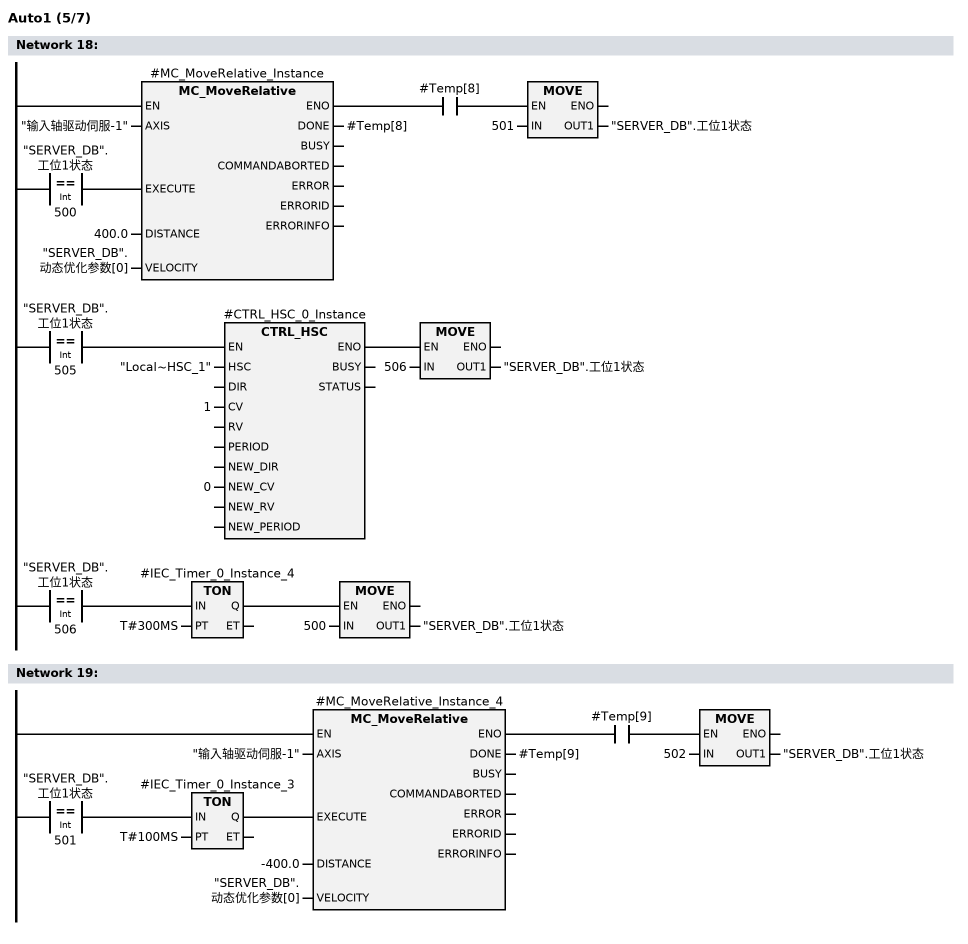
   // ENO of a box is taken as its EN; it also drops when the box reports an error
   #MC_MoveRelative_Instance(Axis := "输入轴驱动伺服-1",   // MC_MoveRelative
                           Execute := "SERVER_DB".工位1状态 = 500,
                           Distance := 400.0,
                           Velocity := "SERVER_DB".动态优化参数[0],
                           Done => #Temp[8]);
   IF #Temp[8] THEN "SERVER_DB".工位1状态 := 501; END_IF;
   #_w1 := "SERVER_DB".工位1状态 = 505;
   IF #_w1 THEN
       #CTRL_HSC_0_Instance(HSC := "Local~HSC_1", CV := 1, NEW_CV := 0);   // CTRL_HSC
       "SERVER_DB".工位1状态 := 506;
   END_IF;
   #IEC_Timer_0_Instance_4(IN := "SERVER_DB".工位1状态 = 506, PT := T#300MS);   // TON
   IF #IEC_Timer_0_Instance_4.Q THEN "SERVER_DB".工位1状态 := 500; END_IF;
END_REGION

REGION Network 19
   // ENO of a box is taken as its EN; it also drops when the box reports an error
   #IEC_Timer_0_Instance_3(IN := "SERVER_DB".工位1状态 = 501, PT := T#100MS);   // TON
   #MC_MoveRelative_Instance_4(Axis := "输入轴驱动伺服-1",   // MC_MoveRelative
                           Execute := #IEC_Timer_0_Instance_3.Q,
                           Distance := -400.0,
                           Velocity := "SERVER_DB".动态优化参数[0],
                           Done => #Temp[9]);
   IF #Temp[9] THEN "SERVER_DB".工位1状态 := 502; END_IF;
END_REGION

REGION Network 20
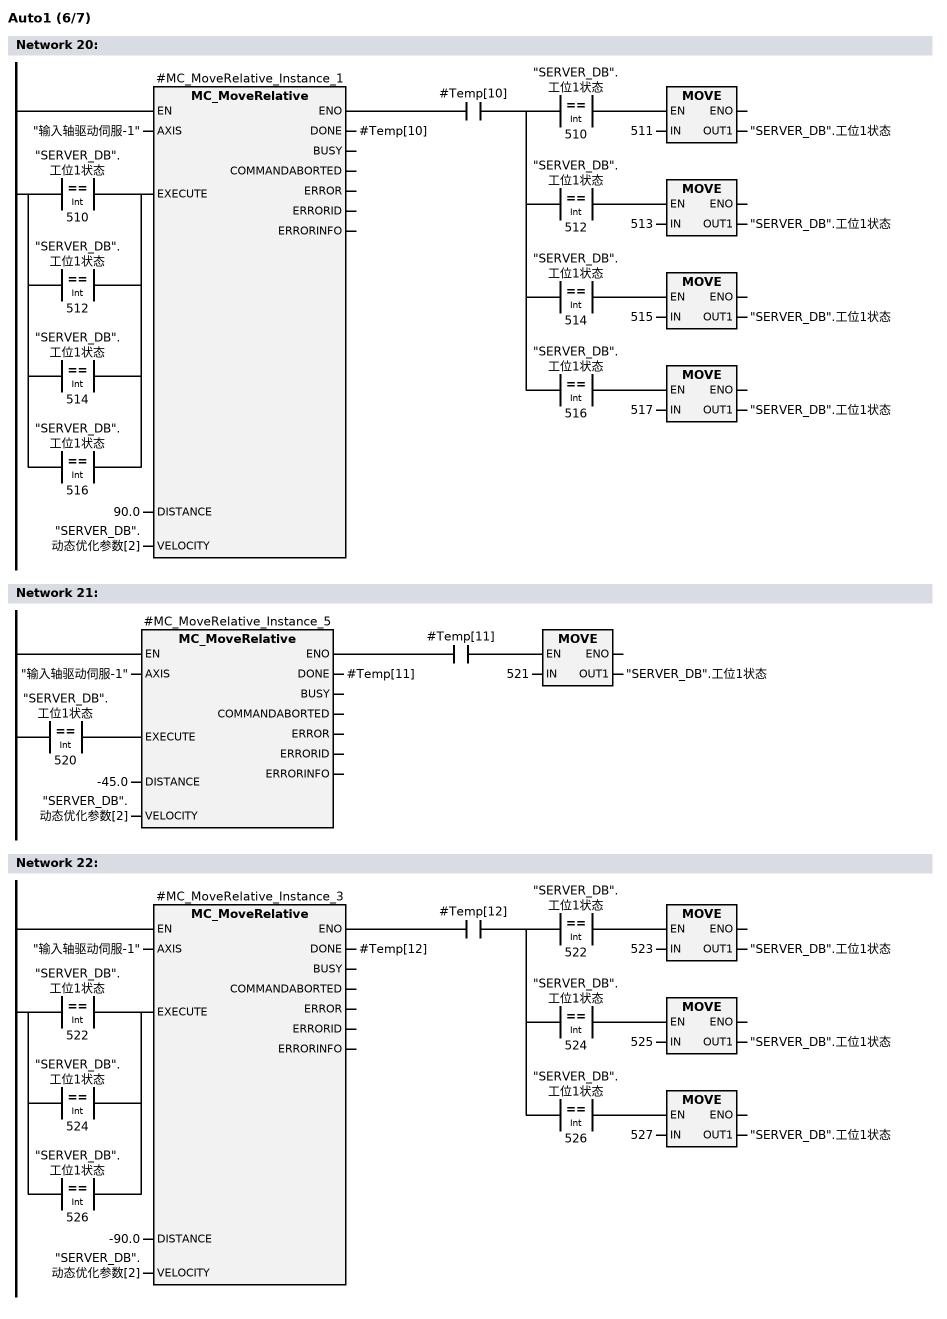
   // ENO of a box is taken as its EN; it also drops when the box reports an error
   #MC_MoveRelative_Instance_1(Axis := "输入轴驱动伺服-1",   // MC_MoveRelative
                           Execute := ("SERVER_DB".工位1状态 = 510) OR ("SERVER_DB".工位1状态 = 512) OR ("SERVER_DB".工位1状态 = 514) OR ("SERVER_DB".工位1状态 = 516),
                           Distance := 90.0,
                           Velocity := "SERVER_DB".动态优化参数[2],
                           Done => #Temp[10]);
   IF #Temp[10] AND ("SERVER_DB".工位1状态 = 510) THEN "SERVER_DB".工位1状态 := 511; END_IF;
   IF #Temp[10] AND ("SERVER_DB".工位1状态 = 512) THEN "SERVER_DB".工位1状态 := 513; END_IF;
   IF #Temp[10] AND ("SERVER_DB".工位1状态 = 514) THEN "SERVER_DB".工位1状态 := 515; END_IF;
   IF #Temp[10] AND ("SERVER_DB".工位1状态 = 516) THEN "SERVER_DB".工位1状态 := 517; END_IF;
END_REGION

REGION Network 21
   // ENO of a box is taken as its EN; it also drops when the box reports an error
   #MC_MoveRelative_Instance_5(Axis := "输入轴驱动伺服-1",   // MC_MoveRelative
                           Execute := "SERVER_DB".工位1状态 = 520,
                           Distance := -45.0,
                           Velocity := "SERVER_DB".动态优化参数[2],
                           Done => #Temp[11]);
   IF #Temp[11] THEN "SERVER_DB".工位1状态 := 521; END_IF;
END_REGION

REGION Network 22
   // ENO of a box is taken as its EN; it also drops when the box reports an error
   #MC_MoveRelative_Instance_3(Axis := "输入轴驱动伺服-1",   // MC_MoveRelative
                           Execute := ("SERVER_DB".工位1状态 = 522) OR ("SERVER_DB".工位1状态 = 524) OR ("SERVER_DB".工位1状态 = 526),
                           Distance := -90.0,
                           Velocity := "SERVER_DB".动态优化参数[2],
                           Done => #Temp[12]);
   IF #Temp[12] AND ("SERVER_DB".工位1状态 = 522) THEN "SERVER_DB".工位1状态 := 523; END_IF;
   IF #Temp[12] AND ("SERVER_DB".工位1状态 = 524) THEN "SERVER_DB".工位1状态 := 525; END_IF;
   IF #Temp[12] AND ("SERVER_DB".工位1状态 = 526) THEN "SERVER_DB".工位1状态 := 527; END_IF;
END_REGION

REGION Network 23
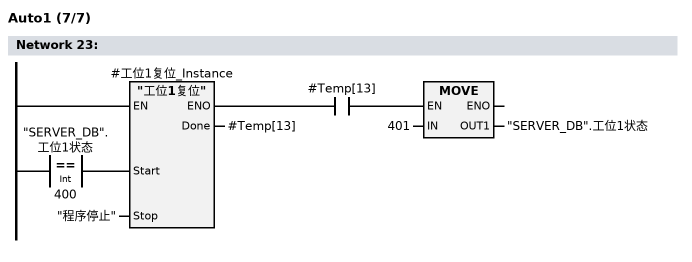
   RUNG wire#powerrail
      #工位1复位_Instance(Start := wire#w1, Stop := "程序停止", Done => #Temp[13])
      Contact( #Temp[13] )
      Move(in := 401, out1 => "SERVER_DB".工位1状态)
   END_RUNG
   RUNG wire#powerrail
      { S7_Templates := "SrcType := Int" } EQ_Contact(in1 := "SERVER_DB".工位1状态, in2 := 400)
   END_RUNG wire#w1
   // the same network as SCL:
   #工位1复位_Instance(Start := "SERVER_DB".工位1状态 = 400, Stop := "程序停止", Done => #Temp[13], ENO => #_w1);   // "工位1复位"
   IF #_w1 AND #Temp[13] THEN "SERVER_DB".工位1状态 := 401; END_IF;
END_REGION
END_FUNCTION_BLOCK

FUNCTION_BLOCK "输入轴二次夹紧"   // FB10, LAD
{ S7_Optimized_Access := 'TRUE' }
VERSION : 0.1
   VAR_INPUT
      Axis : TO_PositioningAxis;
      Start : Bool;
      夹紧位置 : Real;
   END_VAR
   VAR_OUTPUT
      Done : Bool;
   END_VAR
   VAR
      "Step" : Int;
      Temp : Array[0..3] of Bool;
      MC_MoveAbsolute_Instance : MC_MoveAbsolute;
      IEC_Timer_0_Instance : TON_TIME;
      IEC_Timer_0_Instance_1 : TON_TIME;
   END_VAR
   VAR_TEMP   // added for the SCL form of the ladder/FBD networks
      _w1 : Bool;
   END_VAR
BEGIN

REGION Network 1
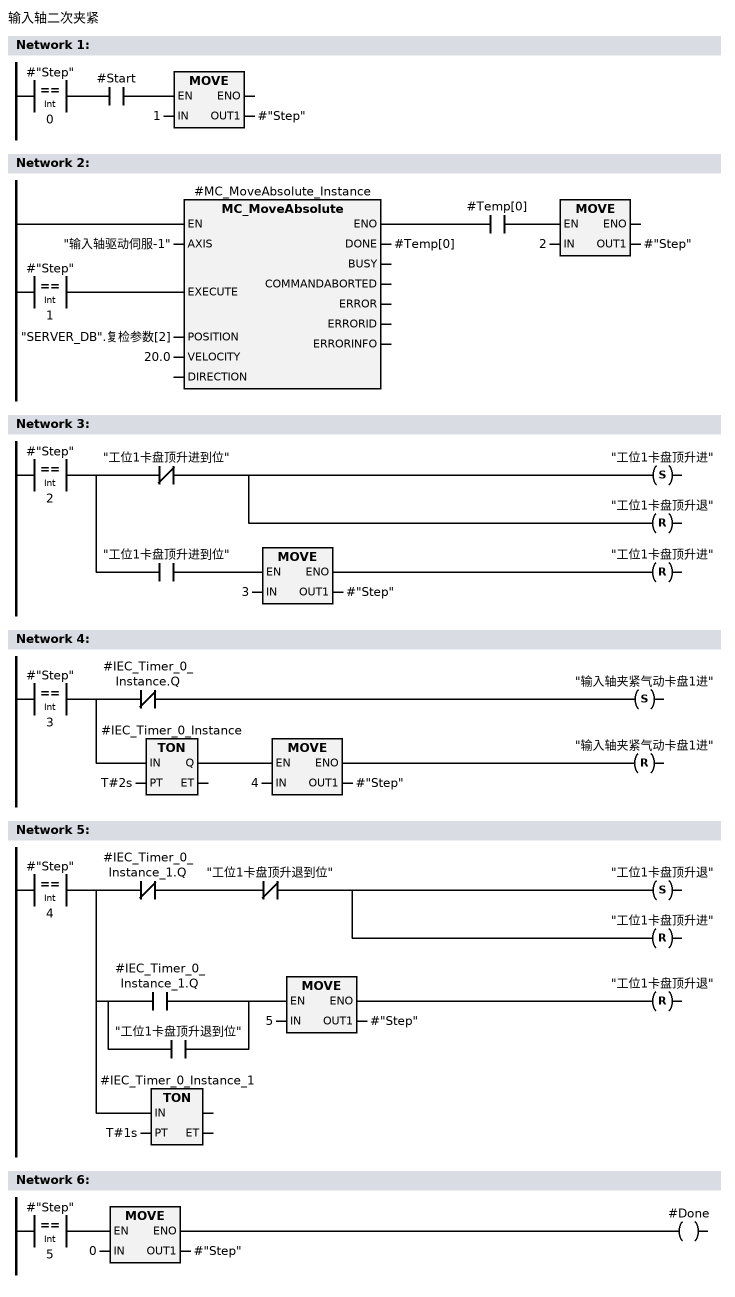
   RUNG wire#powerrail
      { S7_Templates := "SrcType := Int" } EQ_Contact(in1 := #"Step", in2 := 0)
      Contact( #Start )
      Move(in := 1, out1 => #"Step")
   END_RUNG
   // the same network as SCL:
   IF (#"Step" = 0) AND #Start THEN #"Step" := 1; END_IF;
END_REGION

REGION Network 2
   // ENO of a box is taken as its EN; it also drops when the box reports an error
   #MC_MoveAbsolute_Instance(Axis := "输入轴驱动伺服-1",   // MC_MoveAbsolute
                           Execute := #"Step" = 1,
                           Position := "SERVER_DB".复检参数[2],
                           Velocity := 20.0,
                           Done => #Temp[0]);
   IF #Temp[0] THEN #"Step" := 2; END_IF;
END_REGION

REGION Network 3
   RUNG wire#powerrail
      { S7_Templates := "SrcType := Int" } EQ_Contact(in1 := #"Step", in2 := 2)
      wire#w1
      I_Contact( "工位1卡盘顶升进到位" )
      wire#w2
      S_Coil( "工位1卡盘顶升进" )
   END_RUNG
   RUNG wire#w2
      R_Coil( "工位1卡盘顶升退" )
   END_RUNG
   RUNG wire#w1
      Contact( "工位1卡盘顶升进到位" )
      Move(in := 3, out1 => #"Step")
      R_Coil( "工位1卡盘顶升进" )
   END_RUNG
   // the same network as SCL:
   #_w1 := #"Step" = 2;
   IF #_w1 AND NOT "工位1卡盘顶升进到位" THEN
       "工位1卡盘顶升进" := TRUE;
       "工位1卡盘顶升退" := FALSE;
   END_IF;
   IF #_w1 AND "工位1卡盘顶升进到位" THEN
       #"Step" := 3;
       "工位1卡盘顶升进" := FALSE;
   END_IF;
END_REGION

REGION Network 4
   #_w1 := #"Step" = 3;
   IF #_w1 AND NOT #IEC_Timer_0_Instance.Q THEN "输入轴夹紧气动卡盘1进" := TRUE; END_IF;
   #IEC_Timer_0_Instance(IN := #_w1, PT := T#2s);   // TON
   IF #IEC_Timer_0_Instance.Q THEN
       #"Step" := 4;
       "输入轴夹紧气动卡盘1进" := FALSE;
   END_IF;
END_REGION

REGION Network 5
   #_w1 := #"Step" = 4;
   IF #_w1 AND NOT #IEC_Timer_0_Instance_1.Q AND NOT "工位1卡盘顶升退到位" THEN
       "工位1卡盘顶升退" := TRUE;
       "工位1卡盘顶升进" := FALSE;
   END_IF;
   IF #_w1 AND (#IEC_Timer_0_Instance_1.Q OR "工位1卡盘顶升退到位") THEN
       #"Step" := 5;
       "工位1卡盘顶升退" := FALSE;
   END_IF;
   #IEC_Timer_0_Instance_1(IN := #_w1, PT := T#1s);   // TON
END_REGION

REGION Network 6
   RUNG wire#powerrail
      { S7_Templates := "SrcType := Int" } EQ_Contact(in1 := #"Step", in2 := 5)
      Move(in := 0, out1 => #"Step")
      Coil( #Done )
   END_RUNG
   // the same network as SCL:
   #_w1 := #"Step" = 5;
   IF #_w1 THEN #"Step" := 0; END_IF;
   #Done := #_w1;
END_REGION
END_FUNCTION_BLOCK

FUNCTION_BLOCK "输入轴移载夹紧"   // FB11, LAD
{ S7_Optimized_Access := 'TRUE' }
VERSION : 0.1
   VAR_INPUT
      Axis : TO_PositioningAxis;
      接近位置 : Real;
      接近速度 : Real;
      最终位置 : Real;
      最终速度 : Real;
      夹紧 : Bool;
      松开 : Bool;
   END_VAR
   VAR_OUTPUT
      Done : Bool;
   END_VAR
   VAR
      "Step" : Int;
      Temp : Array[0..7] of Bool;
      MC_MoveAbsolute_Instance : MC_MoveAbsolute;
      MC_MoveAbsolute_Instance_1 : MC_MoveAbsolute;
      MC_MoveAbsolute_Instance_2 : MC_MoveAbsolute;
      IEC_Timer_0_Instance : TON_TIME;
      IEC_Timer_0_Instance_1 : TON_TIME;
      MC_MoveAbsolute_Instance_3 : MC_MoveAbsolute;
      MC_MoveAbsolute_Instance_4 : MC_MoveAbsolute;
      MC_MoveAbsolute_Instance_5 : MC_MoveAbsolute;
      IEC_Timer_0_Instance_2 : TON_TIME;
      IEC_Timer_0_Instance_3 : TON_TIME;
      IEC_Timer_0_Instance_4 : TON_TIME;
      MC_MoveRelative_Instance : MC_MoveRelative;
      MC_MoveRelative_Instance_1 : MC_MoveRelative;
   END_VAR
   VAR RETAIN
      IEC_Counter_0_Instance : CTU_INT;
   END_VAR
   VAR_TEMP   // added for the SCL form of the ladder/FBD networks
      _w1 : Bool;
   END_VAR
BEGIN

REGION Network 1
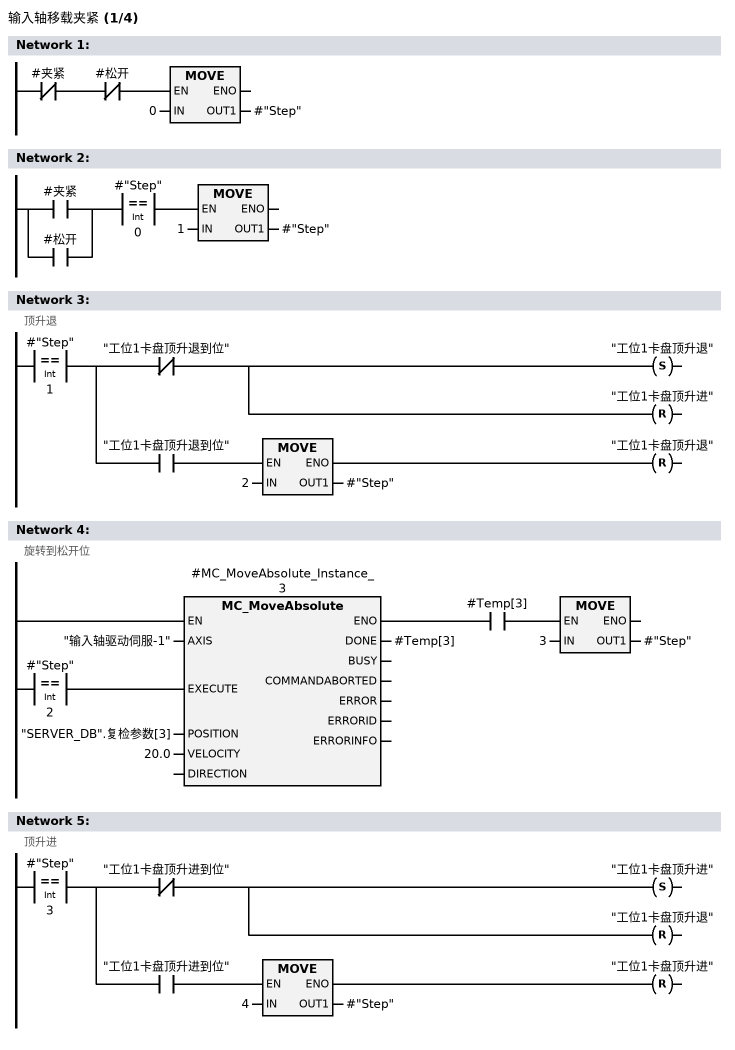
   RUNG wire#powerrail
      I_Contact( #夹紧 )
      I_Contact( #松开 )
      Move(in := 0, out1 => #"Step")
   END_RUNG
   // the same network as SCL:
   IF NOT #夹紧 AND NOT #松开 THEN #"Step" := 0; END_IF;
END_REGION

REGION Network 2
   RUNG wire#powerrail
      Contact( #夹紧 )
      wire#w1
      { S7_Templates := "SrcType := Int" } EQ_Contact(in1 := #"Step", in2 := 0)
      Move(in := 1, out1 => #"Step")
   END_RUNG
   RUNG wire#powerrail
      Contact( #松开 )
   END_RUNG wire#w1
   // the same network as SCL:
   IF (#夹紧 OR #松开) AND (#"Step" = 0) THEN #"Step" := 1; END_IF;
END_REGION

REGION Network 3
   // 顶升退
   RUNG wire#powerrail
      { S7_Templates := "SrcType := Int" } EQ_Contact(in1 := #"Step", in2 := 1)
      wire#w1
      I_Contact( "工位1卡盘顶升退到位" )
      wire#w2
      S_Coil( "工位1卡盘顶升退" )
   END_RUNG
   RUNG wire#w2
      R_Coil( "工位1卡盘顶升进" )
   END_RUNG
   RUNG wire#w1
      Contact( "工位1卡盘顶升退到位" )
      Move(in := 2, out1 => #"Step")
      R_Coil( "工位1卡盘顶升退" )
   END_RUNG
   // the same network as SCL:
   #_w1 := #"Step" = 1;
   IF #_w1 AND NOT "工位1卡盘顶升退到位" THEN
       "工位1卡盘顶升退" := TRUE;
       "工位1卡盘顶升进" := FALSE;
   END_IF;
   IF #_w1 AND "工位1卡盘顶升退到位" THEN
       #"Step" := 2;
       "工位1卡盘顶升退" := FALSE;
   END_IF;
END_REGION

REGION Network 4
   // 旋转到松开位
   // ENO of a box is taken as its EN; it also drops when the box reports an error
   #MC_MoveAbsolute_Instance_3(Axis := "输入轴驱动伺服-1",   // MC_MoveAbsolute
                           Execute := #"Step" = 2,
                           Position := "SERVER_DB".复检参数[3],
                           Velocity := 20.0,
                           Done => #Temp[3]);
   IF #Temp[3] THEN #"Step" := 3; END_IF;
END_REGION

REGION Network 5
   // 顶升进
   RUNG wire#powerrail
      { S7_Templates := "SrcType := Int" } EQ_Contact(in1 := #"Step", in2 := 3)
      wire#w1
      I_Contact( "工位1卡盘顶升进到位" )
      wire#w2
      S_Coil( "工位1卡盘顶升进" )
   END_RUNG
   RUNG wire#w2
      R_Coil( "工位1卡盘顶升退" )
   END_RUNG
   RUNG wire#w1
      Contact( "工位1卡盘顶升进到位" )
      Move(in := 4, out1 => #"Step")
      R_Coil( "工位1卡盘顶升进" )
   END_RUNG
   // the same network as SCL:
   #_w1 := #"Step" = 3;
   IF #_w1 AND NOT "工位1卡盘顶升进到位" THEN
       "工位1卡盘顶升进" := TRUE;
       "工位1卡盘顶升退" := FALSE;
   END_IF;
   IF #_w1 AND "工位1卡盘顶升进到位" THEN
       #"Step" := 4;
       "工位1卡盘顶升进" := FALSE;
   END_IF;
END_REGION

REGION Network 6
   // 卡盘松开
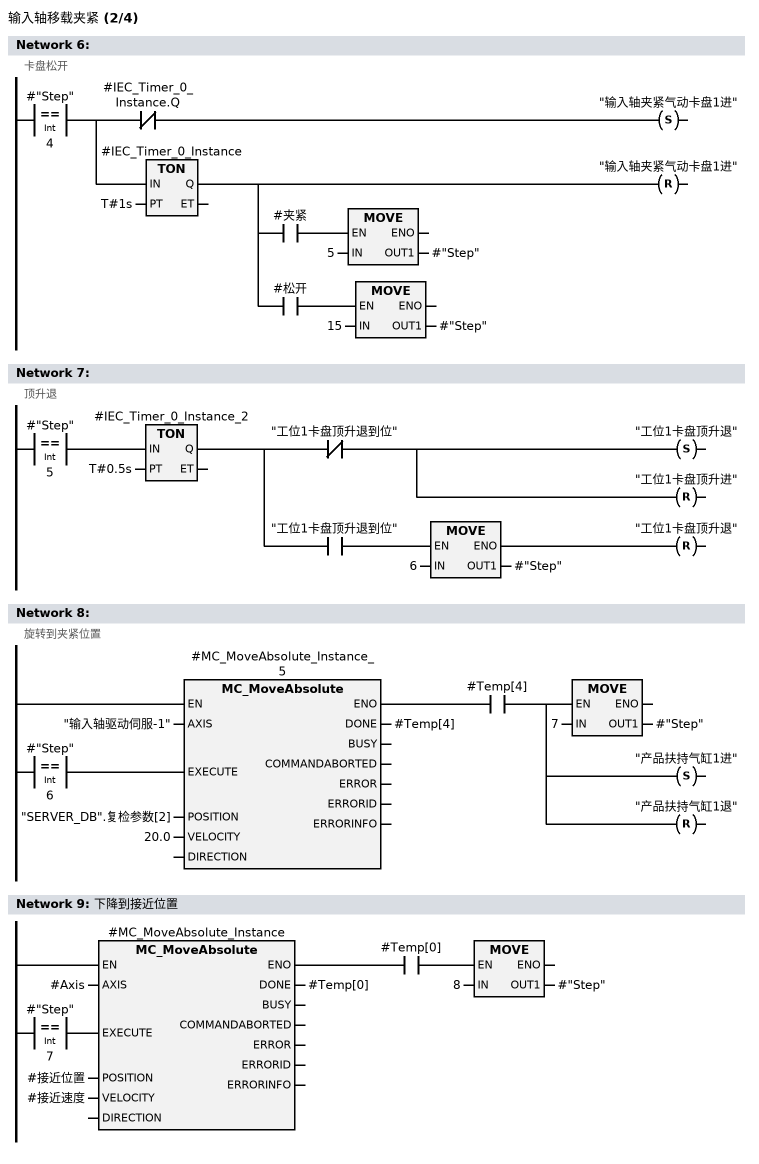
   #_w1 := #"Step" = 4;
   IF #_w1 AND NOT #IEC_Timer_0_Instance.Q THEN "输入轴夹紧气动卡盘1进" := TRUE; END_IF;
   #IEC_Timer_0_Instance(IN := #_w1, PT := T#1s);   // TON
   IF #IEC_Timer_0_Instance.Q THEN "输入轴夹紧气动卡盘1进" := FALSE; END_IF;
   IF #IEC_Timer_0_Instance.Q AND #夹紧 THEN #"Step" := 5; END_IF;
   IF #IEC_Timer_0_Instance.Q AND #松开 THEN #"Step" := 15; END_IF;
END_REGION

REGION Network 7
   // 顶升退
   #IEC_Timer_0_Instance_2(IN := #"Step" = 5, PT := T#0.5s);   // TON
   IF #IEC_Timer_0_Instance_2.Q AND NOT "工位1卡盘顶升退到位" THEN
       "工位1卡盘顶升退" := TRUE;
       "工位1卡盘顶升进" := FALSE;
   END_IF;
   IF #IEC_Timer_0_Instance_2.Q AND "工位1卡盘顶升退到位" THEN
       #"Step" := 6;
       "工位1卡盘顶升退" := FALSE;
   END_IF;
END_REGION

REGION Network 8
   // 旋转到夹紧位置
   // ENO of a box is taken as its EN; it also drops when the box reports an error
   #MC_MoveAbsolute_Instance_5(Axis := "输入轴驱动伺服-1",   // MC_MoveAbsolute
                           Execute := #"Step" = 6,
                           Position := "SERVER_DB".复检参数[2],
                           Velocity := 20.0,
                           Done => #Temp[4]);
   IF #Temp[4] THEN
       #"Step" := 7;
       "产品扶持气缸1进" := TRUE;
       "产品扶持气缸1退" := FALSE;
   END_IF;
END_REGION

REGION Network 9: 下降到接近位置
   // ENO of a box is taken as its EN; it also drops when the box reports an error
   #MC_MoveAbsolute_Instance(Axis := #Axis,   // MC_MoveAbsolute
                           Execute := #"Step" = 7,
                           Position := #接近位置,
                           Velocity := #接近速度,
                           Done => #Temp[0]);
   IF #Temp[0] THEN #"Step" := 8; END_IF;
END_REGION

REGION Network 10: 慢速下降套花键
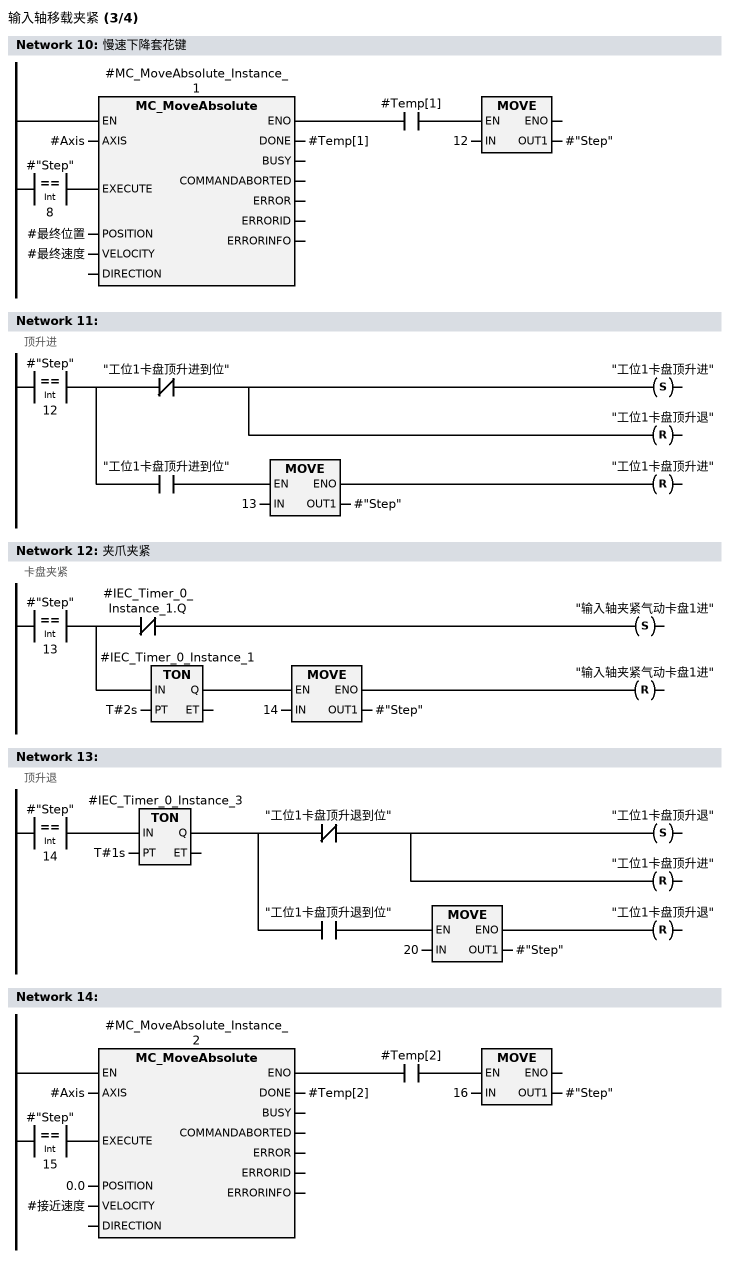
   // ENO of a box is taken as its EN; it also drops when the box reports an error
   #MC_MoveAbsolute_Instance_1(Axis := #Axis,   // MC_MoveAbsolute
                           Execute := #"Step" = 8,
                           Position := #最终位置,
                           Velocity := #最终速度,
                           Done => #Temp[1]);
   IF #Temp[1] THEN #"Step" := 12; END_IF;
END_REGION

REGION Network 11
   // 顶升进
   RUNG wire#powerrail
      { S7_Templates := "SrcType := Int" } EQ_Contact(in1 := #"Step", in2 := 12)
      wire#w1
      I_Contact( "工位1卡盘顶升进到位" )
      wire#w2
      S_Coil( "工位1卡盘顶升进" )
   END_RUNG
   RUNG wire#w2
      R_Coil( "工位1卡盘顶升退" )
   END_RUNG
   RUNG wire#w1
      Contact( "工位1卡盘顶升进到位" )
      Move(in := 13, out1 => #"Step")
      R_Coil( "工位1卡盘顶升进" )
   END_RUNG
   // the same network as SCL:
   #_w1 := #"Step" = 12;
   IF #_w1 AND NOT "工位1卡盘顶升进到位" THEN
       "工位1卡盘顶升进" := TRUE;
       "工位1卡盘顶升退" := FALSE;
   END_IF;
   IF #_w1 AND "工位1卡盘顶升进到位" THEN
       #"Step" := 13;
       "工位1卡盘顶升进" := FALSE;
   END_IF;
END_REGION

REGION Network 12: 夹爪夹紧
   // 卡盘夹紧
   #_w1 := #"Step" = 13;
   IF #_w1 AND NOT #IEC_Timer_0_Instance_1.Q THEN "输入轴夹紧气动卡盘1进" := TRUE; END_IF;
   #IEC_Timer_0_Instance_1(IN := #_w1, PT := T#2s);   // TON
   IF #IEC_Timer_0_Instance_1.Q THEN
       #"Step" := 14;
       "输入轴夹紧气动卡盘1进" := FALSE;
   END_IF;
END_REGION

REGION Network 13
   // 顶升退
   #IEC_Timer_0_Instance_3(IN := #"Step" = 14, PT := T#1s);   // TON
   IF #IEC_Timer_0_Instance_3.Q AND NOT "工位1卡盘顶升退到位" THEN
       "工位1卡盘顶升退" := TRUE;
       "工位1卡盘顶升进" := FALSE;
   END_IF;
   IF #IEC_Timer_0_Instance_3.Q AND "工位1卡盘顶升退到位" THEN
       #"Step" := 20;
       "工位1卡盘顶升退" := FALSE;
   END_IF;
END_REGION

REGION Network 14
   // ENO of a box is taken as its EN; it also drops when the box reports an error
   #MC_MoveAbsolute_Instance_2(Axis := #Axis,   // MC_MoveAbsolute
                           Execute := #"Step" = 15,
                           Position := 0.0,
                           Velocity := #接近速度,
                           Done => #Temp[2]);
   IF #Temp[2] THEN #"Step" := 16; END_IF;
END_REGION

REGION Network 15
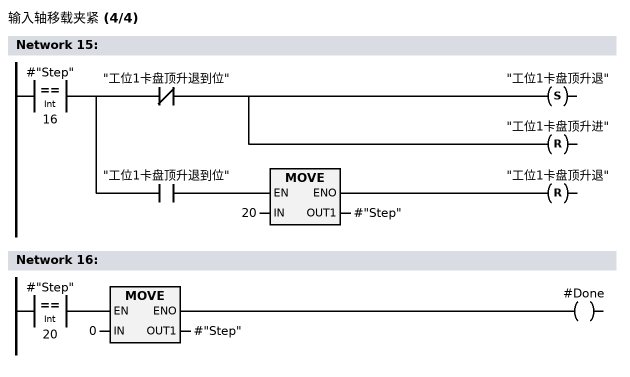
   RUNG wire#powerrail
      { S7_Templates := "SrcType := Int" } EQ_Contact(in1 := #"Step", in2 := 16)
      wire#w1
      I_Contact( "工位1卡盘顶升退到位" )
      wire#w2
      S_Coil( "工位1卡盘顶升退" )
   END_RUNG
   RUNG wire#w2
      R_Coil( "工位1卡盘顶升进" )
   END_RUNG
   RUNG wire#w1
      Contact( "工位1卡盘顶升退到位" )
      Move(in := 20, out1 => #"Step")
      R_Coil( "工位1卡盘顶升退" )
   END_RUNG
   // the same network as SCL:
   #_w1 := #"Step" = 16;
   IF #_w1 AND NOT "工位1卡盘顶升退到位" THEN
       "工位1卡盘顶升退" := TRUE;
       "工位1卡盘顶升进" := FALSE;
   END_IF;
   IF #_w1 AND "工位1卡盘顶升退到位" THEN
       #"Step" := 20;
       "工位1卡盘顶升退" := FALSE;
   END_IF;
END_REGION

REGION Network 16
   RUNG wire#powerrail
      { S7_Templates := "SrcType := Int" } EQ_Contact(in1 := #"Step", in2 := 20)
      Move(in := 0, out1 => #"Step")
      Coil( #Done )
   END_RUNG
   // the same network as SCL:
   #_w1 := #"Step" = 20;
   IF #_w1 THEN #"Step" := 0; END_IF;
   #Done := #_w1;
END_REGION
END_FUNCTION_BLOCK

FUNCTION_BLOCK "动态优化"   // FB12, LAD
{ S7_Optimized_Access := 'TRUE' }
VERSION : 0.1
BEGIN
END_FUNCTION_BLOCK

FUNCTION "Analog To Project amount" : Void   // FC1, LAD
{ S7_Optimized_Access := 'TRUE' }
VERSION : 0.1
   VAR_INPUT
      Analog : Int;
      Min_Value : Real;
      Max_Value : Real;
   END_VAR
   VAR_OUTPUT
      Project_amount : Real;
   END_VAR
   VAR_TEMP
      Temp_Value : Real;
   END_VAR
BEGIN

REGION Network 1
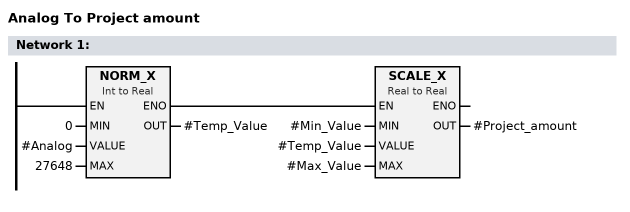
   RUNG wire#powerrail
      { S7_Templates := "[SrcType := Int, DestType := Real]" } Normalize(min := 0, value := #Analog, max := 27648, out => #Temp_Value)
      { S7_Templates := "[SrcType := Real, DestType := Real]" } Scale(min := #Min_Value, value := #Temp_Value, max := #Max_Value, out => #Project_amount)
   END_RUNG
   // the same network as SCL:
   #Temp_Value := NORM_X(MIN := 0, VALUE := #Analog, MAX := 27648);
   #Project_amount := SCALE_X(MIN := #Min_Value, VALUE := #Temp_Value, MAX := #Max_Value);
END_REGION
END_FUNCTION

FUNCTION "encoder" : Void   // FC2, LAD
{ S7_Optimized_Access := 'TRUE' }
VERSION : 0.1
   VAR_INPUT
      encoder : DInt;
   END_VAR
   VAR_OUTPUT
      angle : Real;
   END_VAR
   VAR_TEMP
      Temp_Value : DInt;
      Temp_Value2 : DInt;
   END_VAR
BEGIN

REGION Network 1
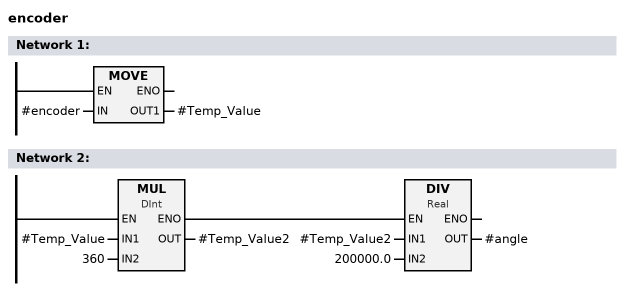
   RUNG wire#powerrail
      Move(in := #encoder, out1 => #Temp_Value)
   END_RUNG
   // the same network as SCL:
   #Temp_Value := #encoder;
END_REGION

REGION Network 2
   RUNG wire#powerrail
      { S7_Templates := "SrcType := DInt" } Mul(in1 := #Temp_Value, in2 := 360, out => #Temp_Value2)
      { S7_Templates := "SrcType := Real" } Div(in1 := #Temp_Value2, in2 := 200000.0, out => #angle)
   END_RUNG
   // the same network as SCL:
   #Temp_Value2 := #Temp_Value * 360;
   #angle := #Temp_Value2 / 200000.0;
END_REGION
END_FUNCTION

ORGANIZATION_BLOCK "Main"   // OB1, LAD, ProgramCycle
TITLE = "Main Program Sweep (Cycle)"
{ S7_Optimized_Access := 'TRUE' }
VERSION : 0.1
   VAR_INPUT
      Initial_Call : Bool;   // Initial call of this OB
      Remanence : Bool;   // =True, if remanent data are available
   END_VAR
   VAR_TEMP   // added for the SCL form of the ladder/FBD networks
      _w1 : Bool;
   END_VAR
BEGIN

REGION Network 1
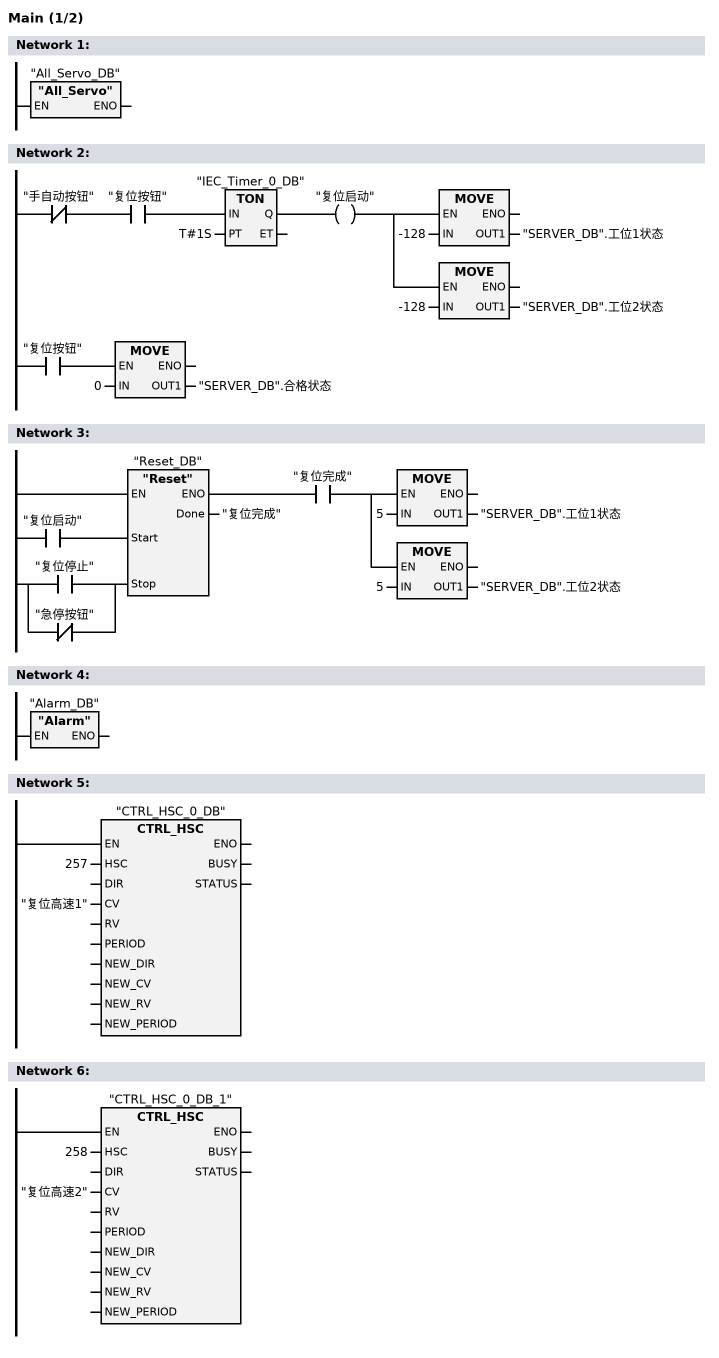
   RUNG wire#powerrail
      "All_Servo_DB"()
   END_RUNG
   // the same network as SCL:
   "All_Servo_DB"();   // "All_Servo"
END_REGION

REGION Network 2
   "IEC_Timer_0_DB".TON(IN := NOT "手自动按钮" AND "复位按钮", PT := T#1S);
   "复位启动" := "IEC_Timer_0_DB".Q;
   IF "IEC_Timer_0_DB".Q THEN
       "SERVER_DB".工位1状态 := -128;
       "SERVER_DB".工位2状态 := -128;
   END_IF;
   IF "复位按钮" THEN "SERVER_DB".合格状态 := 0; END_IF;
END_REGION

REGION Network 3
   RUNG wire#powerrail
      "Reset_DB"(Start := wire#w1, Stop := wire#w2, Done => "复位完成")
      Contact( "复位完成" )
      wire#w3
      Move(in := 5, out1 => "SERVER_DB".工位1状态)
   END_RUNG
   RUNG wire#powerrail
      Contact( "复位启动" )
   END_RUNG wire#w1
   RUNG wire#powerrail
      Contact( "复位停止" )
   END_RUNG wire#w2
   RUNG wire#powerrail
      I_Contact( "急停按钮" )
   END_RUNG wire#w2
   RUNG wire#w3
      Move(in := 5, out1 => "SERVER_DB".工位2状态)
   END_RUNG
   // the same network as SCL:
   "Reset_DB"(Start := "复位启动", Stop := "复位停止" OR NOT "急停按钮", Done => "复位完成", ENO => #_w1);   // "Reset"
   IF #_w1 AND "复位完成" THEN
       "SERVER_DB".工位1状态 := 5;
       "SERVER_DB".工位2状态 := 5;
   END_IF;
END_REGION

REGION Network 4
   RUNG wire#powerrail
      "Alarm_DB"()
   END_RUNG
   // the same network as SCL:
   "Alarm_DB"();   // "Alarm"
END_REGION

REGION Network 5
   "CTRL_HSC_0_DB"(HSC := 257, CV := "复位高速1");   // CTRL_HSC
END_REGION

REGION Network 6
   "CTRL_HSC_0_DB_1"(HSC := 258, CV := "复位高速2");   // CTRL_HSC
END_REGION

REGION Network 7
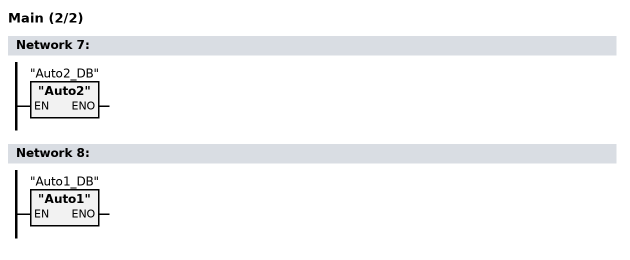
   RUNG wire#powerrail
      "Auto2_DB"()
   END_RUNG
   // the same network as SCL:
   "Auto2_DB"();   // "Auto2"
END_REGION

REGION Network 8
   RUNG wire#powerrail
      "Auto1_DB"()
   END_RUNG
   // the same network as SCL:
   "Auto1_DB"();   // "Auto1"
END_REGION
END_ORGANIZATION_BLOCK

ORGANIZATION_BLOCK "Cyclic interrupt"   // OB30, LAD, CyclicInterrupt
{ S7_Optimized_Access := 'TRUE' }
VERSION : 0.1
   VAR_INPUT
      Initial_Call : Bool;   // Initial call of this OB
      Event_Count : Int;   // Events discarded
   END_VAR
   VAR_TEMP   // added for the SCL form of the ladder/FBD networks
      _w1 : Bool;
   END_VAR
BEGIN

REGION Network 1
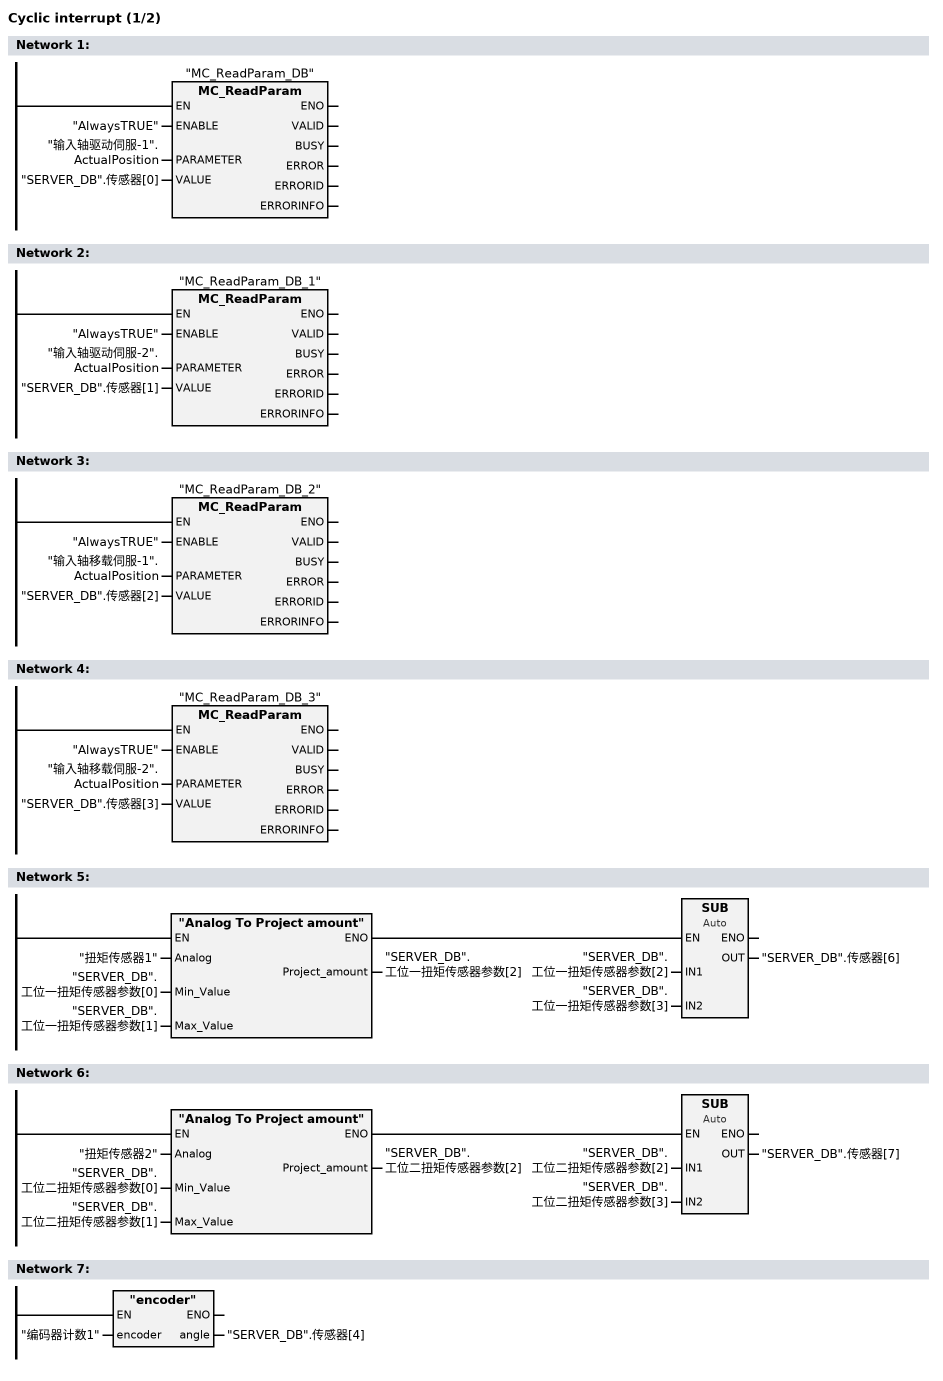
   "MC_ReadParam_DB"(Enable := "AlwaysTRUE",   // MC_ReadParam
                     Parameter := "输入轴驱动伺服-1".ActualPosition,
                     Value := "SERVER_DB".传感器[0]);
END_REGION

REGION Network 2
   "MC_ReadParam_DB_1"(Enable := "AlwaysTRUE",   // MC_ReadParam
                       Parameter := "输入轴驱动伺服-2".ActualPosition,
                       Value := "SERVER_DB".传感器[1]);
END_REGION

REGION Network 3
   "MC_ReadParam_DB_2"(Enable := "AlwaysTRUE",   // MC_ReadParam
                       Parameter := "输入轴移载伺服-1".ActualPosition,
                       Value := "SERVER_DB".传感器[2]);
END_REGION

REGION Network 4
   "MC_ReadParam_DB_3"(Enable := "AlwaysTRUE",   // MC_ReadParam
                       Parameter := "输入轴移载伺服-2".ActualPosition,
                       Value := "SERVER_DB".传感器[3]);
END_REGION

REGION Network 5
   RUNG wire#powerrail
      "Analog To Project amount"(Analog := "扭矩传感器1", Min_Value := "SERVER_DB".工位一扭矩传感器参数[0], Max_Value := "SERVER_DB".工位一扭矩传感器参数[1], Project_amount => "SERVER_DB".工位一扭矩传感器参数[2])
      Sub(in1 := "SERVER_DB".工位一扭矩传感器参数[2], in2 := "SERVER_DB".工位一扭矩传感器参数[3], out => "SERVER_DB".传感器[6])
   END_RUNG
   // the same network as SCL:
   "Analog To Project amount"(Analog := "扭矩传感器1",
                           Min_Value := "SERVER_DB".工位一扭矩传感器参数[0],
                           Max_Value := "SERVER_DB".工位一扭矩传感器参数[1],
                           Project_amount => "SERVER_DB".工位一扭矩传感器参数[2],
                           ENO => #_w1);
   IF #_w1 THEN "SERVER_DB".传感器[6] := "SERVER_DB".工位一扭矩传感器参数[2] - "SERVER_DB".工位一扭矩传感器参数[3]; END_IF;
END_REGION

REGION Network 6
   RUNG wire#powerrail
      "Analog To Project amount"(Analog := "扭矩传感器2", Min_Value := "SERVER_DB".工位二扭矩传感器参数[0], Max_Value := "SERVER_DB".工位二扭矩传感器参数[1], Project_amount => "SERVER_DB".工位二扭矩传感器参数[2])
      Sub(in1 := "SERVER_DB".工位二扭矩传感器参数[2], in2 := "SERVER_DB".工位二扭矩传感器参数[3], out => "SERVER_DB".传感器[7])
   END_RUNG
   // the same network as SCL:
   "Analog To Project amount"(Analog := "扭矩传感器2",
                           Min_Value := "SERVER_DB".工位二扭矩传感器参数[0],
                           Max_Value := "SERVER_DB".工位二扭矩传感器参数[1],
                           Project_amount => "SERVER_DB".工位二扭矩传感器参数[2],
                           ENO => #_w1);
   IF #_w1 THEN "SERVER_DB".传感器[7] := "SERVER_DB".工位二扭矩传感器参数[2] - "SERVER_DB".工位二扭矩传感器参数[3]; END_IF;
END_REGION

REGION Network 7
   RUNG wire#powerrail
      "encoder"(encoder := "编码器计数1", angle => "SERVER_DB".传感器[4])
   END_RUNG
   // the same network as SCL:
   "encoder"(encoder := "编码器计数1", angle => "SERVER_DB".传感器[4]);
END_REGION

REGION Network 8
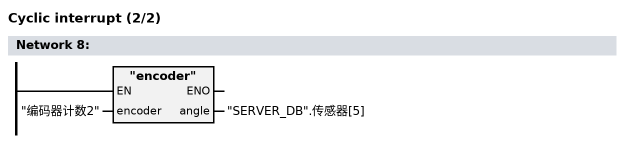
   RUNG wire#powerrail
      "encoder"(encoder := "编码器计数2", angle => "SERVER_DB".传感器[5])
   END_RUNG
   // the same network as SCL:
   "encoder"(encoder := "编码器计数2", angle => "SERVER_DB".传感器[5]);
END_REGION
END_ORGANIZATION_BLOCK